FUNCTION_BLOCK FB_ReadAlias
VAR_INPUT
	bExecute : BOOL := FALSE;
	slv_addr : UINT := 0;
END_VAR
VAR_OUTPUT
	state : INT := 0;
	bError : BOOL;
	value : UDINT := 0;
	
END_VAR
VAR
	fbSdoRead : FB_EcCoESdoRead;
	nErrID : UDINT :=0;
	sdo_address: UINT := 16#8008;
	subIndex: BYTE := 1;
	
END_VAR

fbSdoRead(
        sNetId          := MAIN.sNetId_local,
        //nSlaveAddr      := nSlaveAddr,
		nSlaveAddr :=   slv_addr,
        nIndex          := sdo_address,
        nSubIndex       := subIndex,
        pDstBuf         := ADR(value),
        cbBufLen        := SIZEOF(value),
        bExecute        := bExecute
);
state := 1;
IF NOT fbSdoRead.bBusy THEN
        bExecute := FALSE;
		//done	:= TRUE;
        IF NOT fbSdoRead.bError THEN 
                (* write successful *)
                bError := FALSE;
                nErrId := 0;
        ELSE 
                (* write failed *)
                bError := fbSdoRead.bError;
                nErrId := fbSdoRead.nErrId;
        END_IF
        fbSdoRead(bExecute := FALSE);
		state := 0;
END_IF

END_FUNCTION_BLOCK

(* stored: Version 1.1.0.1, ProductVersion 3.1.4024.10
   POU FB_ReadAlias: Id {7ee7d4eb-decb-4234-923d-9407643d4a01}, SpecialFunc None *)
